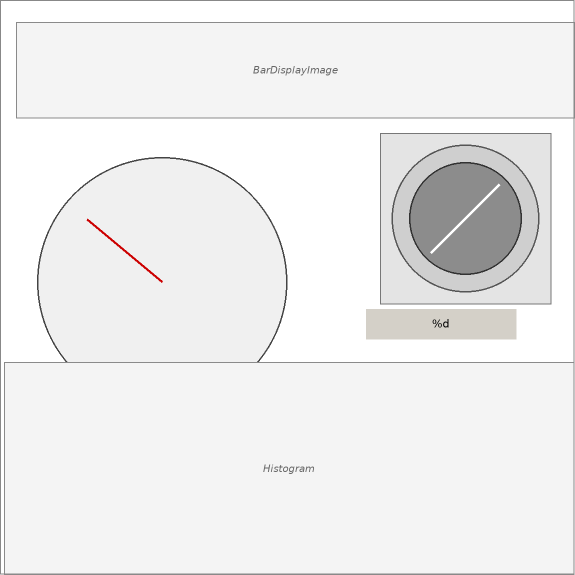
VISUALIZATION P02_Measurement  // 575x575
    BarDisplayImage (16,22 559x96), value: Main.iValueBarDisplay, style: BarDisplayImage-Gray, scale format: %.1f, scale 0..1000
    Meter180 (37,157 250x250), value: Main.iValueBarDisplay, style: Meter-Meter180-Gray, scale format: %.1f, scale 0..1000
    Potentiometer360 (362,133 207x171), variable: Main.bValuePotentialMeter, style: Potentiometer-Potentiometer360-Gray, scale format: %.1f, scale 0..100
        p2431819421: Outside
    Textfield (366,309 150x30), "%d", text variable: Main.bValuePotentialMeter
    Histogram (4,362 570x213), scale format: %.1f, scale 0..1
        p1518820177: Main.aryLrSin
        p102497268: Main.aryLrSin
        p788070771: ARRAY [0..200] OF LREAL
END_VISUALIZATION

(* stored: Version 1.1.0.1, ProductVersion 3.1.4024.4
   Visu P02_Measurement: Id {f4a710b7-b189-450f-93e7-b5a64db82f38} *)
